PROGRAM pouS1Prompts
VAR
	


idbMsgPrompt: FB_CheckMessageBounds;
END_VAR

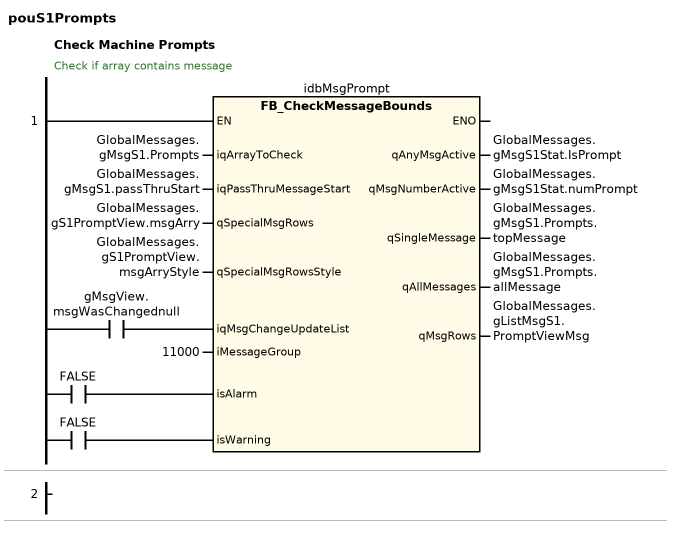
// NETWORK 1: Check Machine Prompts
// Check if array contains message
idbMsgPrompt(
    iqArrayToCheck := GlobalMessages.gMsgS1.Prompts,
    iqPassThruMessageStart := GlobalMessages.gMsgS1.passThruStart,
    qSpecialMsgRows := GlobalMessages.gS1PromptView.msgArry,
    qSpecialMsgRowsStyle := GlobalMessages.gS1PromptView.msgArryStyle,
    iqMsgChangeUpdateList := gMsgView.msgWasChangednull,
    iMessageGroup := 11000,
    isAlarm := FALSE,
    isWarning := FALSE,
    qAnyMsgActive => GlobalMessages.gMsgS1Stat.IsPrompt,
    qMsgNumberActive => GlobalMessages.gMsgS1Stat.numPrompt,
    qSingleMessage => GlobalMessages.gMsgS1.Prompts.topMessage,
    qAllMessages => GlobalMessages.gMsgS1.Prompts.allMessage,
    qMsgRows => GlobalMessages.gListMsgS1.PromptViewMsg); // FB_CheckMessageBounds

// NETWORK 2

END_PROGRAM

(* stored: Version 1.1.0.1, ProductVersion 3.1.4024.11
   POU pouS1Prompts: Id {d0bcea03-d9bc-4b96-baec-8989514f2c5f}, SpecialFunc None *)
